(*
SPDX-FileCopyrightText: © 2026 Oleksandr Tiutyk <trofimich@gmail.com>
SPDX-License-Identifier: MIT
License: https://opensource.org/license/mit
*)

(*!
<summary>Provides FIFO insertion and destructive head removal.</summary>
<description>
Successful insertion transfers disposal responsibility for owned payload; borrowed payload must remain alive
while stored. The caller-side descriptor copy is not reset and must not be released again after transfer.
Independent owning aliases and overlapping owned allocations are unsupported. Peek borrows the head;
RemoveFirst releases it rather than transferring it to the caller. Clear releases owned payload and dynamic
backing storage.
</description>
*)

INTERFACE IQueue EXTENDS IReadOnlyQueue

(*!
<summary>Removes all entries and releases dynamic backing storage.</summary>
<description>
Owned payload is released best effort through GENERIC_VALUE.Release; borrowed storage is not freed. Static
capacity and the borrowed validator are retained. Dynamic capacity becomes zero. Returns this collection and
invalidates positions and views. Cleanup callbacks must not reenter mutation.
</description>
*)
METHOD Clear : IQueue
END_METHOD

(*!
<summary>Copies a value and appends it to the FIFO tail.</summary>
<description>
Borrows the original during the call. isObject = TRUE requires a live Object FB instance implementing
ICloneable; other data is copied as bytes without recursively cloning references. A prepared copy is released
if insertion fails before acceptance; exceptions propagate. Engine-managed exception objects are unsupported.
The original exception is captured before prepared-copy cleanup, so nested cleanup handling cannot replace
its payload. Terminal OOM takes precedence; capture failure still attempts prepared-copy disposal.
</description>
*)
METHOD EnqueueCopy : IQueue
VAR_INPUT
	value : ANY;
	isObject : BOOL := FALSE;
END_VAR
END_METHOD

(*!
<summary>Appends a descriptor after the FIFO tail.</summary>
<description>
Successful insertion transfers disposal responsibility for owned payload; borrowed payload must remain alive
while stored. The caller-side descriptor copy is not reset and must not be released again after transfer.
Independent owning aliases and overlapping owned allocations are unsupported. Full static storage raises an
exception. A configured validator is invoked once before any capacity growth or ownership acceptance.
Validation failure leaves the buffer, Length and incoming ownership unchanged; its exception propagates.
Validator callbacks must not mutate this collection.
</description>
*)
METHOD EnqueueGeneric : IQueue
VAR_INPUT
	value : TOF_Core.GENERIC_VALUE;
END_VAR
END_METHOD

(*!
<summary>Removes the FIFO head without transferring it to the caller.</summary>
<description>
An empty queue raises CollectionEmptyException. Owned head storage is released best effort, not returned to
the caller. Remaining descriptors shift left in linear time. Returns this queue; positions and views may
change. Cleanup callbacks must not reenter mutation.
</description>
*)
METHOD RemoveFirst : IQueue
END_METHOD

(*!
<summary>Exposes the configured value validator.</summary>
<description>
Borrowed optional reference fixed at initialization. Zero means no validator. The collection does not own or
release it.
</description>
*)
{attribute 'monitoring' := 'call'}
PROPERTY ValueValidator : TOF_Core.IGenericValueValidator
GET
END_GET
END_PROPERTY

END_INTERFACE

(* stored: Version 1.1.0.1
   Itf IQueue: Id {134f0e5a-305a-452c-bd7c-b09cb743ac75}
   Method Clear: Id {10bc2c98-bbdf-4b17-a361-6d54bc2adcc2}
   Method EnqueueCopy: Id {c28d5910-db64-43ef-8934-1cf48c41b5c1}
   Method EnqueueGeneric: Id {6f687203-d2e0-4504-a951-6321be6916e4}
   Method RemoveFirst: Id {aa7e88f2-8409-4011-9a0c-cfd3873c980a}
   Property ValueValidator: Id {77f7ebc2-e636-4ab7-a9ea-b7bb22cd07df}
   Get Get: Id {6f03c27d-882e-43e5-89ac-e62962783cb1} *)
